TYPE ST_CircuitBreakerOperationRecord :
STRUCT
    dtTimestamp: DATE_AND_TIME;                 // İşlem zamanı
    eOperation: E_CircuitBreakerPosition;       // İşlem tipi (ON/OFF/TRIPPED)
    eControlMode: E_CircuitBreakerControlMode;  // Kontrol modu
    eFaultCode: E_CircuitBreakerFault;          // Arıza kodu (varsa)
    nBreakerID: INT;                            // Kesici ID
END_STRUCT
END_TYPE

(* stored: Version 1.1.0.1, ProductVersion 3.1.4024.15
   DUT ST_CircuitBreakerOperationRecord: Id {bd5b0ebd-9971-4329-bd21-8c15e7188330} *)
